% RSLogix 500 project blower HOA.RSS, saved by version 8.30.00.16 %
PROJECT "UNTITLED"    % processor: Bul.1763 MicroLogix 1100 Series B %

PROGRAM FILES
  LAD 2 "MAIN"  3 rungs
  LAD 4 "DIGITALI/O"  5 rungs
  LAD 5 "CONTROLS"  5 rungs

DATA FILES
  O0 OUTPUT  5 elements
  I1 INPUT  7 elements
  S2 STATUS  66 elements
  B3 BINARY  1 elements
  T4 TIMER  1 elements
  C5 COUNTER  1 elements
  R6 CONTROL  1 elements
  N7 INTEGER  1 elements
  F8 FLOAT  1 elements

LADDER 2 "MAIN"
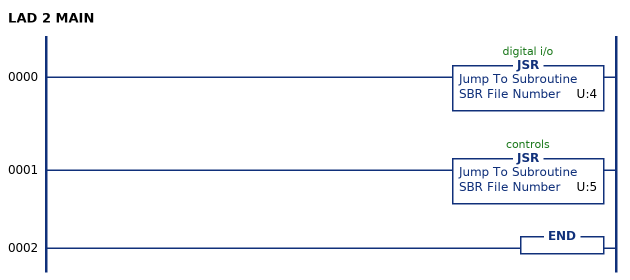
% Rung: 0 %
SOR JSR U:4 EOR
%   U:4  "digital i/o" %
% Rung: 1 %
SOR JSR U:5 EOR
%   U:5  "controls" %
% Rung: 2 %
SOR END EOR

LADDER 4 "DIGITALI/O"
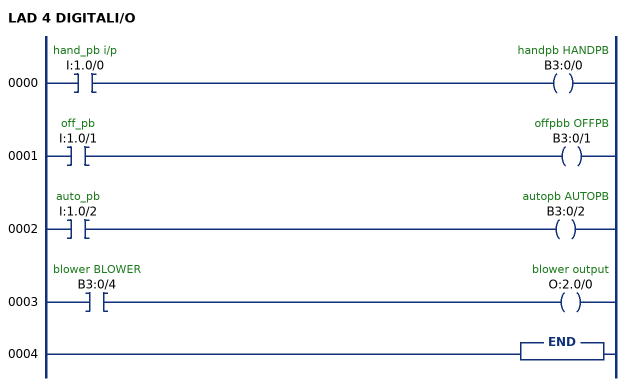
% Rung: 0 %
SOR XIC I:1.0/0 OTE B3:0/0 EOR
%   I:1.0/0  "hand_pb i/p" %
%   B3:0/0  HANDPB  "handpb" %
% Rung: 1 %
SOR XIC I:1.0/1 OTE B3:0/1 EOR
%   I:1.0/1  "off_pb" %
%   B3:0/1  OFFPB  "offpbb" %
% Rung: 2 %
SOR XIC I:1.0/2 OTE B3:0/2 EOR
%   I:1.0/2  "auto_pb" %
%   B3:0/2  AUTOPB  "autopb" %
% Rung: 3 %
SOR XIC B3:0/4 OTE O:2.0/0 EOR
%   B3:0/4  BLOWER  "blower" %
%   O:2.0/0  "blower output" %
% Rung: 4 %
SOR END EOR

LADDER 5 "CONTROLS"
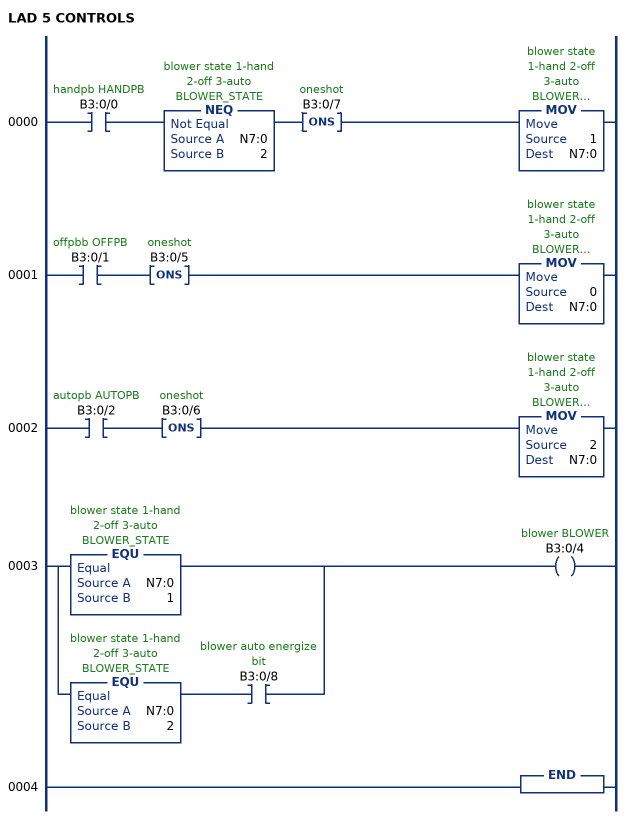
% Rung: 0 %
SOR XIC B3:0/0 NEQ N7:0 2 ONS B3:0/7 MOV 1 N7:0 EOR
%   B3:0/0  HANDPB  "handpb" %
%   N7:0  BLOWER_STATE  "blower state 1-hand 2-off 3-auto" %
%   B3:0/7  "oneshot" %
% Rung: 1 %
SOR XIC B3:0/1 ONS B3:0/5 MOV 0 N7:0 EOR
%   B3:0/1  OFFPB  "offpbb" %
%   B3:0/5  "oneshot" %
%   N7:0  BLOWER_STATE  "blower state 1-hand 2-off 3-auto" %
% Rung: 2 %
SOR XIC B3:0/2 ONS B3:0/6 MOV 2 N7:0 EOR
%   B3:0/2  AUTOPB  "autopb" %
%   B3:0/6  "oneshot" %
%   N7:0  BLOWER_STATE  "blower state 1-hand 2-off 3-auto" %
% Rung: 3 %
SOR BST EQU N7:0 1 NXB EQU N7:0 2 XIC B3:0/8 BND OTE B3:0/4 EOR
%   N7:0  BLOWER_STATE  "blower state 1-hand 2-off 3-auto" %
%   B3:0/8  "blower auto energize bit" %
%   B3:0/4  BLOWER  "blower" %
% Rung: 4 %
SOR END EOR
